FUNCTION_BLOCK Button_NO
VAR
	_input AT%M*	:BOOL;
END_VAR

PROPERTY IsPressed : BOOL
GET
IsPressed:= _input;
END_GET
END_PROPERTY

END_FUNCTION_BLOCK

(* stored: Version 1.1.0.1, ProductVersion 3.1.4024.12
   POU Button_NO: Id {6a31ca67-2efd-4a12-9b08-d9d7ccb5fe91}, SpecialFunc None
   Property IsPressed: Id {41f3700b-46e7-499b-ba0c-97c1c152ff2d}
   Get Get: Id {4b486152-cfe4-4136-b2da-a2c8f67032f3} *)
